// TwinCAT 3 PLC project Main
// ProgramVersion: 3.1.4024.0
// libraries:
//   Tc2_Standard, * (Beckhoff Automation GmbH)
//   Tc2_System, * (Beckhoff Automation GmbH)
//   Tc2_Utilities, * (Beckhoff Automation GmbH)
//   Tc3_JsonXml, * (Beckhoff Automation GmbH)
//   Tc3_Module, * (Beckhoff Automation GmbH)
//   TcUnit, * (www.tcunit.org)
//   mobject-core,0.4.0,mobject
//   mobject-server,0.14.0,mobject
// project tree:
//   / Param.TcGVL, PlcTask.TcTTO
//   POUs/ MAIN.TcPOU
//   Tests/Mocks/ AdjustableSizeReplyRpcHandler.TcPOU, RejectWithMessageSyncHandler.TcPOU, SyncToAsyncEchoRpcHandler.TcPOU, RejectWithMessageAsyncHandler.TcPOU
//   Tests/ Server_IntegrationTestSuite.TcPOU
//   Tests/_Internal/ ChunkedRequestData_TestSuite.TcPOU (not stored)
// real-time tasks:
//   TASK PlcTask: cycle T#10ms, priority 20, ADS port 350

CONFIGURATION Main
    RESOURCE PLC ON TwinCAT3
        TASK PlcTask(INTERVAL := T#10ms, PRIORITY := 20);
        PROGRAM MAIN WITH PlcTask : MAIN;
    END_RESOURCE
END_CONFIGURATION

// ---- Param.TcGVL
{attribute 'qualified_only'}
VAR_GLOBAL CONSTANT
	test : BOOL := true;
END_VAR

// ---- POUs/MAIN.TcPOU
PROGRAM MAIN
VAR
	server_IntegrationTestSuite : Server_IntegrationTestSuite;
	chunkedRequestData_TestSuite : ChunkedRequestData_TestSuite;
	
	initialized : BOOL;
	server : RpcServer;
	concatStringRpcHandler : ConcatStringRpcHandler;	
	syncToAsyncEchoRpcHandler : SyncToAsyncEchoRpcHandler;
	adjustableSizeReplyRpcHandler : AdjustableSizeReplyRpcHandler;
	
END_VAR

TcUnit.RUN();

// the code below is used by TwinCAT HMI implementation

IF NOT initialized THEN
	initialized := TRUE;
	server.RegisterSynchronousRpcHandler('concat',concatStringRpcHandler);
	server.RegisterSynchronousRpcHandler('asyncEcho',syncToAsyncEchoRpcHandler);
	server.RegisterSynchronousRpcHandler('adjustableSizeReply',adjustableSizeReplyRpcHandler);
END_IF

server.CyclicCall();

// this has timers inside, so must be cyclic called.
syncToAsyncEchoRpcHandler.CyclicCall();

END_PROGRAM

// ---- Tests/Server_IntegrationTestSuite.TcPOU
FUNCTION_BLOCK Server_IntegrationTestSuite EXTENDS TcUnit.FB_TestSuite
VAR
	// variables for TestAsyncEchoRpcCallAndResponse
	testAsyncEchoRpcCallAndResponseSetup : BOOL;
	testAsyncEchoRpcCallAndResponseServer : RpcServer;
	testAsyncEchoRpcCallAndResponseAsyncEchoRpcHandler : AsyncEchoRpcHandler;
	testAsyncEchoRpcCallAndResponseOutput : ResponseData;
	
	// variables for TestConcatRpcCallAndResponse
	testConcatRpcCallAndResponseOutput : ResponseData;
	
	// variables for TestAsyncConcatRpcCallAndResponse
	testAsyncConcatRpcCallAndResponseOutput : ResponseData;
END_VAR

//TestSyncToAsyncEchoRpcCallAndResponse();
TestConcatRpcCallAndResponse();
TestConcatRpcCallAndResponseWithChunkedRequest();
TestAsyncConcatRpcCallAndResponse();

METHOD TestAsyncConcatRpcCallAndResponse
VAR
	server : RpcServer;
	asyncConcatStringRpcHandler : AsyncConcatStringRpcHandler;
	header : T_MAXSTRING := '{"Type":"RPC 1.0","Method-Name":"concat","Content-Type":"application/json"}';
    payload : T_MAXSTRING := '{"STR1":"hello", "STR2":"world"}';
	followupHeader : T_MAXSTRING := '{"Type":"RPC 1.0","Accept":"application/json","Method-Name":"asyncEcho","Response-Id":"1","Session-Id":"1"}';
	followupPayload : T_MAXSTRING := '';
	expected : T_MAXSTRING := '"helloworld"';
	actual : T_MAXSTRING;
END_VAR
TEST('TestAsyncConcatRpcCallAndResponse');

server.RegisterAsynchronousRpcHandler('concat',asyncConcatStringRpcHandler);

testAsyncConcatRpcCallAndResponseOutput := server.HandleRequest(header,payload);
server.CyclicCall();
testAsyncConcatRpcCallAndResponseOutput := server.HandleRequest(followupHeader, followupPayload);
actual := testAsyncConcatRpcCallAndResponseOutput.Payload;

AssertEquals(
	Expected := expected, 
	Actual := actual,
	Message := 'Did not produce the expected result'
);

TEST_FINISHED();
END_METHOD

METHOD TestConcatRpcCallAndResponse
VAR
	server : RpcServer;
	concatStringRpcHandler : ConcatStringRpcHandler;
	header : T_MAXSTRING := '{"Type":"RPC 1.0","Method-Name":"concat","Content-Type":"application/json"}';
    payload : T_MAXSTRING := '{"STR1":"hello", "STR2":"world"}';
	expected : T_MAXSTRING := '"helloworld"';
	actual : T_MAXSTRING;
END_VAR
TEST('TestConcatRpcCallAndResponse');

server.RegisterSynchronousRpcHandler('concat',concatStringRpcHandler);

testConcatRpcCallAndResponseOutput := server.HandleRequest(header,payload);
actual := testConcatRpcCallAndResponseOutput.Payload;

AssertEquals(
	Expected := expected, 
	Actual := actual,
	Message := 'Did not produce the expected result'
);

TEST_FINISHED();
END_METHOD

METHOD TestConcatRpcCallAndResponseWithChunkedRequest
VAR
	server : RpcServer;
	concatStringRpcHandler : ConcatStringRpcHandler;
	chunk1Header : T_MAXSTRING := '{"Type":"RPC 1.0","Method-Name":"concat","Request-Id":"abc","Has-More-Chunks":true, "Chunk-Sequence":1, "Chunk-Total":2, "Content-Type":"application/json"}';
    chunk1payload : T_MAXSTRING := '{"STR1":"hello",';
	chunk2Header : T_MAXSTRING := '{"Type":"RPC 1.0","Session-Id":"1","Method-Name":"concat","Request-Id":"abc","Has-More-Chunks":false, "Chunk-Sequence":2, "Chunk-Total":2, "Content-Type":"application/json"}';
    chunk2payload : T_MAXSTRING := ' "STR2":"world"}';
	expected : T_MAXSTRING := '"helloworld"';
	out : ResponseData;
END_VAR
//TEST('TestConcatRpcCallAndResponseWithChunkedRequest');

//server.RegisterRpcHandler('concat',concatStringRpcHandler);

//out := server.HandleRequest(chunk1Header,chunk1payload);
//out := server.HandleRequest(chunk2Header,chunk2payload);

//AssertTrue(
//	Condition := expected = out.Payload,
//	Message := 'Did not produce the expected result'
//);

//TEST_FINISHED();
END_METHOD

METHOD TestSyncToAsyncEchoRpcCallAndResponse
VAR
	header : T_MAXSTRING := '{"Type":"RPC 1.0","Accept":"application/json","Method-Name":"asyncEcho","Content-Type":"application/json"}';
    payload : T_MAXSTRING := '{"Echo":"hello"}';
	followupHeader : T_MAXSTRING := '{"Type":"RPC 1.0","Accept":"application/json","Method-Name":"asyncEcho","Response-Id":"1","Session-Id":"1"}';
	followuPayload : T_MAXSTRING := '{"Echo":"hello"}';
	expected : T_MAXSTRING := '"hello"';
	actual : T_MAXSTRING;
END_VAR
TEST('TestAsyncEchoRpcCallAndResponse');

IF NOT testAsyncEchoRpcCallAndResponseSetup THEN
	testAsyncEchoRpcCallAndResponseServer.RegisterSynchronousRpcHandler('asyncEcho',testAsyncEchoRpcCallAndResponseAsyncEchoRpcHandler);
	testAsyncEchoRpcCallAndResponseOutput := testAsyncEchoRpcCallAndResponseServer.HandleRequest(header,payload);
	testAsyncEchoRpcCallAndResponseSetup := TRUE;	
END_IF

testAsyncEchoRpcCallAndResponseAsyncEchoRpcHandler.CyclicCall();

IF testAsyncEchoRpcCallAndResponseAsyncEchoRpcHandler.Busy THEN
	RETURN;
END_IF

testAsyncEchoRpcCallAndResponseOutput := testAsyncEchoRpcCallAndResponseServer.HandleRequest(followupHeader,followuPayload);
actual := testAsyncEchoRpcCallAndResponseOutput.Payload;

AssertEquals(
	Expected := expected, 
	Actual := actual,
	Message := 'Did not produce the expected result'
);

TEST_FINISHED();
END_METHOD

END_FUNCTION_BLOCK

// ---- Tests/Mocks/SyncToAsyncEchoRpcHandler.TcPOU
FUNCTION_BLOCK SyncToAsyncEchoRpcHandler IMPLEMENTS I_SynchronousRpcHandler
VAR
	asyncResponse : I_AsynchronousRpcResponse;
	result : T_MAXSTRING;
	timer : TON;
END_VAR

PROPERTY PUBLIC Busy : BOOL
GET
Busy := asyncResponse <> 0;
END_GET
END_PROPERTY

METHOD PUBLIC CyclicCall
VAR_INPUT
END_VAR
timer(in := Busy, pt := T#1S);

IF timer.Q THEN
	asyncResponse.CompleteWithString(result);
	asyncResponse := 0;
	result := '';
END_IF
END_METHOD

METHOD Handle
VAR_INPUT
	Parameters : I_Deserializer;
	Response : I_SynchronousRpcResponse;
END_VAR
VAR
	deserializerFeedback : DeserializerFeedback;
	echo : T_MAXSTRING;
END_VAR
IF Busy THEN
	Response.RejectWithMessage('Already processing response');
	RETURN;
END_IF

IF NOT Parameters.TryGetKeyString('Echo', echo, deserializerFeedback) THEN
	Response.RejectWithMessage('Missing Echo parameter');
	RETURN;
END_IF

result := echo;
Response.TryMakeAsynchronous(asyncResponse);
END_METHOD

END_FUNCTION_BLOCK

// ---- Tests/Mocks/AdjustableSizeReplyRpcHandler.TcPOU
FUNCTION_BLOCK AdjustableSizeReplyRpcHandler IMPLEMENTS I_SynchronousRpcHandler
VAR
END_VAR

METHOD Handle
VAR_INPUT
	Parameters : I_Deserializer;
	Response : I_SynchronousRpcResponse;
END_VAR
VAR
	deserializerFeedback : DeserializerFeedback;
	size : UDINT;
	pBytes : POINTER TO BYTE;
	currentPos : POINTER TO BYTE;
	i : UDINT;
	count : BYTE;
END_VAR
IF NOT Parameters.TryGetKeyUdint('Size', size, deserializerFeedback) THEN
	Response.RejectWithMessage('Missing Size parameter');
	RETURN;
END_IF

IF size = 0 THEN 
	Response.CompleteWithNull();
END_IF

pBytes := __NEW(BYTE, size);
FOR i := 0 TO size -1 DO
	currentPos := pBytes + i;
	currentPos^ := count;
	count := count + 1;
END_FOR

Response.CompleteWithBytesAsHex(pBytes, size);

__Delete(pBytes);
END_METHOD

END_FUNCTION_BLOCK

// ---- Tests/Mocks/RejectWithMessageSyncHandler.TcPOU
FUNCTION_BLOCK RejectWithMessageSyncHandler IMPLEMENTS I_SynchronousRpcHandler
VAR
END_VAR

METHOD Handle
VAR_INPUT
	Parameters : I_Deserializer;
	Response : I_SynchronousRpcResponse;
END_VAR
VAR
END_VAR
Response.RejectWithMessage('This is the reject message');
END_METHOD

END_FUNCTION_BLOCK

// ---- Tests/Mocks/RejectWithMessageAsyncHandler.TcPOU
FUNCTION_BLOCK RejectWithMessageAsyncHandler IMPLEMENTS I_AsynchronousRpcHandler
VAR
END_VAR

METHOD Handle
VAR_INPUT
	Parameters : I_Deserializer;
	Response : I_AsynchronousRpcResponse;
END_VAR
VAR
END_VAR
Response.RejectWithMessage('This is the reject message');
END_METHOD

END_FUNCTION_BLOCK
